//------------------------------------------------------------------------------------------
//                                                                                        	
//***************************** Beckhoff TwinCAT Examples **********************************
//                                                                                        	
//************************************* WARNING ********************************************
// This program is only an example. If it is used as a control program in any real        	
// application, Beckhoff is not responsible for any malfunction, loss or damage           	
// which could arise by using this program!                                               	
//                                                                                        	
//*************************************  Program Info. *************************************
//                                                                                        	
// PLC program name:       	F_Replace (Function)               	                           	
// Software platform:      	TwinCat v3.1.4024.10
//							Database Server 3.3.33.1				                          	
// Modified by:            	Per Søgaard Carlsen 			                                  	
// Email:					p.carlsen@beckhoff.com	                                  	
//                                                                                        	
// ======================================================================================== 
//         Version       Date                        Remarks                              	
// ======================================================================================== 
//         1.0           10 july 2020                 First release of this example        	
// ======================================================================================== 
//                                                                                        	
//******************************* Aims OF this PLC PROGRAM *********************************
//                                                                                        	
// Execute SQL quires in expert mode						 			                             
//                                                                                        	
//-----------------------------------------------------------------------------------------

FUNCTION_BLOCK FB_EasySql

VAR_INPUT
	bExecute : BOOL;
	wDBID : WORD; //DBID
	pSql : POINTER TO BYTE; //Pointer to SQL command string
	cbSql : UDINT; //Sizeof of SSql command string
	pData : POINTER TO BYTE; //Pointer to data array to store readed data from database - set to 0 for write
	cbData : UDINT; //Sizeof data array for stored data.  - set to 0 for write
	udiMaxOfRecord : UDINT; //Maximum numbers of data record to read.
END_VAR
	
VAR_OUTPUT
	udiNoOfRecords : UDINT; //Hvor mange record er fundet
	bDone : BOOL; //Database skrivning afsluttet
	bBusy : BOOL; //Database skrivning afsluttet
	bError : BOOL; //Fejl under skrivning til database
	sError : STRING(255); //Fejl beskrivelse
END_VAR

VAR
	fbSqlConnection : FB_SQLDatabaseEvt(sNetID:='',tTimeout:=T#5S);
	fbSqlCommand : FB_SQLCommandEvt(sNetID:='',tTimeout:=T#5S);
	fbSqlResult : FB_SQLResultEvt(sNetID:='', tTimeout   := T#5S);
	iState : INT;
	ipResultEvent : Tc3_Eventlogger.I_TcMessage;
	bInternDone : BOOL;
	bInternError : BOOL;
END_VAR

CASE iState OF
	0:
		
		IF bExecute THEN //Whait for start
			bBusy := TRUE;
			M_Zero();
			iState := 100;
		END_IF
					
	100: //Open database connection

		fbSqlConnection.Connect(hDBID:= wDBID);
				
		IF NOT fbSqlConnection.bBusy THEN
			IF fbSqlConnection.bError THEN
				ipResultEvent := fbSqlConnection.ipTcResult;
				iState := 9000;	
			ELSE
				iState := 110;	
			END_IF
		END_IF
				
	110: //Init SQL command
											
		IF fbSqlConnection.CreateCmd(ADR(fbSqlCommand)) THEN
			IF fbSqlConnection.bError THEN
				ipResultEvent := fbSqlConnection.ipTcResult;
				iState := 9000;
			ELSE
				IF pData = 0 OR cbData = 0 OR udiMaxOfRecord = 0 THEN
					iState := 130;	
				ELSE
					iState := 120;
				END_IF
				
			END_IF
		END_IF		
				
	120: //Execute SQL command, with data return
			
		IF fbSqlCommand.ExecuteDataReturn(pSQLCmd:=pSql , cbSQLCmd:= cbSql, pSQLDBResult:= ADR(fbSQLResult)) THEN
			ipResultEvent := fbSqlCommand.ipTcResult;
				
			IF udiMaxOfRecord < 1 THEN // Minimum read one record
				udiMaxOfRecord := 1;
			END_IF
					
						
			IF fbSqlResult.Read(0, udiMaxOfRecord, pData, cbData, TRUE, TRUE) THEN //Parse sql data to struct
				IF fbSqlResult.bError THEN
					ipResultEvent := fbSqlResult.ipTcResult;
					udiNoOfRecords := 0;
					iState := 9000; 
				ELSE
					// Data found without any errors
					udiNoOfRecords := fbSqlResult.nDataCount; 
					bInternDone := TRUE;
					iState := 1000; 
				END_IF
			END_IF
			
		END_IF
		
	130: //Execute SQL command, without data return
		IF fbSqlCommand.Execute(pSQLCmd:= pSql, cbSQLCmd:= cbSql) THEN
			IF fbSqlCommand.bError THEN
				ipResultEvent := fbSqlCommand.ipTcResult;
				udiNoOfRecords := 0;
				iState := 9000; 
			ELSE
				// Write data without any errors
				udiNoOfRecords := fbSqlResult.nDataCount; 
				bInternDone := TRUE;
				iState := 1000; 
			END_IF
		END_IF
				
	1000: //Close database connection
		fbSqlConnection.Disconnect();	
		IF NOT fbSqlConnection.bBusy THEN
			iState := 1010;
		END_IF
			
	1010: // Return to start
		bBusy := FALSE;
		bDone := bInternDone;
		bError := bInternError;
		IF NOT bExecute THEN
			bDone := FALSE;
			iState := 0;
		END_IF
								
	9000: //Parse error description
		bInternError := TRUE;
		IF ipResultEvent.RequestEventText(nLangId:= 1033, sResult:= sError, nResultSize:= SIZEOF(sError), bError=> , hrErrorCode=> ) THEN
			iState := 1000;
		END_IF
	
END_CASE

METHOD PRIVATE M_Zero : BOOL
VAR_INPUT
END_VAR
sError := '';
bBusy := FALSE;
bError := FALSE;
bInternError := FALSE;
bDone := FALSE;
bInternDone := FALSE;
udiNoOfRecords := 0;
END_METHOD

END_FUNCTION_BLOCK

(* stored: Version 1.1.0.1, ProductVersion 3.1.4024.4
   POU FB_EasySql: Id {36f86a88-9a01-423b-821d-919b9bd9a854}, SpecialFunc None
   Method M_Zero: Id {50ea0aed-0550-41c0-a44c-7272fd88c4e5} *)
